Fanuc KAREL source: kt00409.KL

-- PROVISIONAL review KL for V1013-1; original PC SHA256 8392ee411cd0cf5b8669a520b5e1b9b7d14a32a1835a153406ebf8513c859bae
-- Incomplete behavior may be omitted. Consult companion uncertainty JSON. Do not deploy.
PROGRAM KT00409
%NOLOCKGROUP
VAR
  B1 : BOOLEAN
  B2 : BOOLEAN
  OUT : BOOLEAN
BEGIN
  -- UNRESOLVED_PC offsets 5-12; opcodes 9D,23
  -- UNRESOLVED_PC offsets 17-24; opcodes 9C,23
  -- UNRESOLVED_PC offsets 29-36; opcodes 9D,23
  -- UNRESOLVED_PC offsets 41-48; opcodes 9C,23
  -- UNRESOLVED_PC offsets 53-72; opcodes 21,21,5B,23
  -- UNRESOLVED_PC offsets 77-81; opcodes 7F
END KT00409
